FUNCTION_BLOCK EventLogger 
VAR
	EventBuffer	:	ARRAY[1..100] OF ST_Event; // Stores events, event buffer
	CurrentEventBufferIndex	:	INT := 0;
	
	_PersistentEventStorage	:	I_PersistentEventStorage;
END_VAR
VAR CONSTANT
	MAXIMUM_SIZE_OF_EVENT_BUFFER	:	INT := 100;
END_VAR

(* True for successful add, false for full buffer*)
METHOD PUBLIC AddEvent : BOOL
VAR_INPUT
	eEventType		: E_EventType;
	eEventSeverity	:	TcEventSeverity;
	nEventIdentity	:	UDINT;
	sEventText		:	STRING(255);
END_VAR
IF NOT IsEventBufferFull() THEN
	CurrentEventBufferIndex := CurrentEventBufferIndex + 1;
	EventBuffer[CurrentEventBufferIndex].eEventType := eEventType;
	EventBuffer[CurrentEventBufferIndex].eEventSeverity := eEventSeverity;
	EventBuffer[CurrentEventBufferIndex].nEventIdentity := nEventIdentity;
	EventBuffer[CurrentEventBufferIndex].sEventText := sEventText;
	UpdateEventTimestampWithSystemTime(stEvent := EventBuffer[CurrentEventBufferIndex]);

	AddEvent := TRUE;
ELSE
	AddEvent := FALSE;
END_IF

// store event persistently
_PersistentEventStorage.StoreEvent(stEvent := EventBuffer[CurrentEventBufferIndex]);
END_METHOD

METHOD FB_Init : BOOL
VAR_INPUT
	bInitRetains	:	BOOL; // if true, retain variables are initialised (warm / cold start)
	bInCopyCode		:	BOOL; // if true, instance after gets moved into the copy code (online change)
	iPersistentEventStorage		:	I_PersistentEventStorage;
END_VAR
_PersistentEventStorage := iPersistentEventStorage;
END_METHOD

METHOD IsEventBufferFull : BOOL
VAR_INPUT
END_VAR
IF (CurrentEventBufferIndex + 1) > MAXIMUM_SIZE_OF_EVENT_BUFFER THEN
	IsEventBufferFull := TRUE;
END_IF
END_METHOD

END_FUNCTION_BLOCK

(* stored: Version 1.1.0.1, ProductVersion 3.1.4024.12
   POU EventLogger: Id {d1982c32-abf0-4cb5-8e3e-ffc59e7bb657}, SpecialFunc None
   Method AddEvent: Id {d3b24734-2908-4dcf-b36e-f2fa37caa4d0}
   Method FB_Init: Id {1a83c867-327a-4af8-b1d8-1d2278bdb361}
   Method IsEventBufferFull: Id {d59e34e1-e8cf-4e3f-b153-c4a82a1fb98c} *)
